FUNCTION_BLOCK AE_AX_CLIENT_0_SUBSCRIBE_1 (* Trigger a remote OPC-UA method call via CLIENT_0 and read the resulting state back via SUBSCRIBE_1, driven by an AE_AX bidirectional adapter Socket (1 Event forward, state back) *)
  (* Standard: 61499-2; Description: Copyright (c) 2026 HR Agrartechnik GmbH This program and the accompanying materials are made available under the terms of the Eclipse Public License 2.0 which is available at https://www.eclipse.org/legal/epl-2.0/ SPDX-License-Identifier: EPL-2.0 *)
  (* Version 1.0, 2026-09-03, Franz Höpfinger, HR Agrartechnik GmbH, initial API and implementation and/or initial documentation *)
  PACKAGE adapter::net;
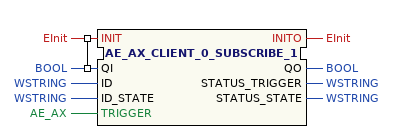
  EVENT_INPUT
    INIT : EInit WITH QI; (* Initialization *)
  END_EVENT
  EVENT_OUTPUT
    INITO : EInit; (* Initialization Confirm *)
  END_EVENT
  VAR_INPUT
    QI : BOOL;
    ID : WSTRING; (* Remote-Methodenadresse fuer den Trigger-Aufruf *)
    ID_STATE : WSTRING; (* Lokal ueberwachter Zustandsknoten (ACTION=READ) *)
  END_VAR
  VAR_OUTPUT
    QO : BOOL; (* TRUE nur wenn CLIENT_0_1 und STATE_SUBSCRIBE aktuell beide QO=TRUE melden *)
    STATUS_TRIGGER : WSTRING; (* STATUS von CLIENT_0_1 *)
    STATUS_STATE : WSTRING; (* STATUS von STATE_SUBSCRIBE *)
  END_VAR
  SOCKETS
    TRIGGER : adapter::types::bidirectional::AE_AX; (* Trigger (out), Zustand (in) *)
  END_SOCKETS
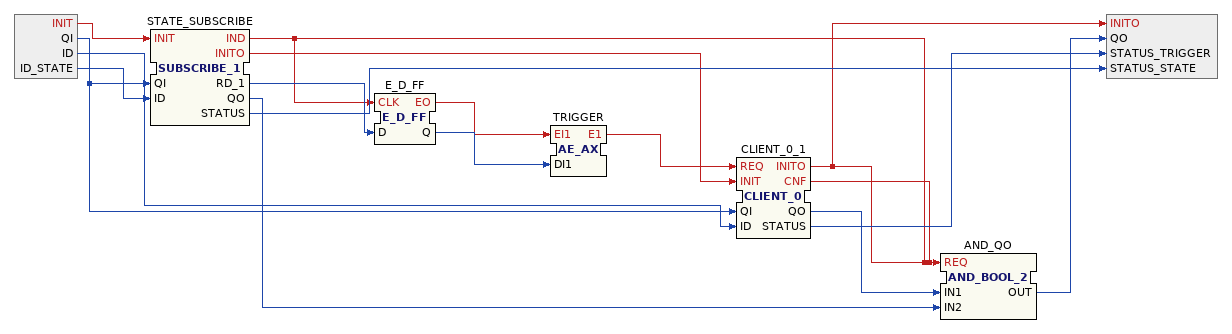
  FBS
    CLIENT_0_1 : iec61499::net::CLIENT_0;
    STATE_SUBSCRIBE : iec61499::net::SUBSCRIBE_1;
    E_D_FF : iec61499::events::E_D_FF;
    AND_QO : iec61131::booleanOperators::AND_BOOL_2;
  END_FBS
  EVENT_CONNECTIONS
    INIT TO STATE_SUBSCRIBE.INIT;
    CLIENT_0_1.INITO TO INITO;
    CLIENT_0_1.INITO TO AND_QO.REQ;
    TRIGGER.E1 TO CLIENT_0_1.REQ;
    STATE_SUBSCRIBE.IND TO E_D_FF.CLK;
    E_D_FF.EO TO TRIGGER.EI1;
    STATE_SUBSCRIBE.INITO TO CLIENT_0_1.INIT;
    CLIENT_0_1.CNF TO AND_QO.REQ;
    STATE_SUBSCRIBE.IND TO AND_QO.REQ;
  END_CONNECTIONS
  DATA_CONNECTIONS
    QI TO CLIENT_0_1.QI;
    QI TO STATE_SUBSCRIBE.QI;
    ID TO CLIENT_0_1.ID;
    ID_STATE TO STATE_SUBSCRIBE.ID;
    STATE_SUBSCRIBE.RD_1 TO E_D_FF.D;
    E_D_FF.Q TO TRIGGER.DI1;
    CLIENT_0_1.QO TO AND_QO.IN1;
    STATE_SUBSCRIBE.QO TO AND_QO.IN2;
    AND_QO.OUT TO QO;
    CLIENT_0_1.STATUS TO STATUS_TRIGGER;
    STATE_SUBSCRIBE.STATUS TO STATUS_STATE;
  END_CONNECTIONS
END_FUNCTION_BLOCK
